PROGRAM GCC1
VAR
END_VAR

// NETWORK 1

END_PROGRAM

(* stored: Version 1.1.0.1, ProductVersion 3.1.4022.3
   POU GCC1: Id {f47a0c78-0e42-4e98-9ce8-4680ec83b10a}, SpecialFunc None *)
